(* IEC 61131-3 sources: CodesysTest/alpha/export/FBs/Components/Temp Sensors/FB_TemperatureSensor.pou/TempReadingC.prop, 1 file *)

(* ---- Get.pm.st ---- *)
(*#-#-#-#-#-#-#-#-#-#---Declaration---#-#-#-#-#-#-#-#-#-#-#-#-#*)

VAR
END_VAR
(*#-#-#-#-#-#-#-#-#-#---Implementation---#-#-#-#-#-#-#-#-#-#-#-#-#*)

TempReadingC := _temperatureReadingC;
